{library PUBLIC}
TYPE ABB_STATUS_OPERATING_MODE :
(
	ABB_STATUS_OPERATION_UNDEF:=0,				(* Undefined operating mode *)
	ABB_STATUS_OPERATION_AUTO:=1,				(* Automatic operating mode *)
	ABB_STATUS_OPERATION_MAN_PROG:=2, 			(* Manual operating mode MAX. 250 mm/S *)
	ABB_STATUS_OPERATION_MAN_TEST:=3 			(* Manual operating mode full speed, 100 % *)
);
END_TYPE

(* stored: Version 1.1.0.1, ProductVersion 3.1.4022.12
   EnumerationTextList ABB_STATUS_OPERATING_MODE: Id {f811a0bb-bce8-4ff7-9cb0-2067f5b2b0cd} *)
